(* Logix 5000 project; controller Machine_Smothies_V0 vendor 1 type 14 code 149 rev 36.11; software revision 36.00 *)

TASK MainTask (continuous, watchdog 500 ms) : MainProgram

MODULES
   Local : vendor 1 type 14 code 149 (Compact 0, rev 36.11)
      Discrete_IO : Embedded (Compact 1, rev 3.1, Output RPI 20 ms)
END_MODULES

VAR_GLOBAL   (* controller tags *)
   Acai : BOOL;
   Acai_Quant_1 : BOOL;
   Acai_Quant_2 : BOOL;
   Acai_Quant_3 : BOOL;
   Ajouter_Verre_Grand : BOOL;
   Ajouter_Verre_Moyen : BOOL;
   Ajouter_Verre_Petit : BOOL;
   Annuler_Base : BOOL;
   Annuler_Choix_Verre : BOOL;
   Annuler_Fruits : BOOL;
   Annuler_Lait : BOOL;
   Annuler_Sucrer : BOOL;
   Annuler_Tout : BOOL;
   Application_Lait : BOOL;
   Application_Sucre : BOOL;
   Avocat : BOOL;
   Avocat_Quant_1 : BOOL;
   Avocat_Quant_2 : BOOL;
   Avocat_Quant_3 : BOOL;
   Banane : BOOL;
   Banane_Quant_1 : BOOL;
   Banane_Quant_2 : BOOL;
   Banane_Quant_3 : BOOL;
   Bleuet : BOOL;
   Bleuet_Quant_1 : BOOL;
   Bleuet_Quant_2 : BOOL;
   Bleuet_Quant_3 : BOOL;
   Capteu_Sucrer : BOOL;
   Capteur_Base : BOOL;
   Capteur_Fruits : BOOL;
   Capteur_Grand : BOOL;
   Capteur_Lait : BOOL;
   Capteur_Moyen : BOOL;
   Capteur_Petit : BOOL;
   Capteur_Preparer : BOOL;
   Capteur_Pret : BOOL := 1;
   Choix_Verre_Grand : BOOL;
   Choix_Verre_Moyen : BOOL;
   Choix_Verre_Petit : BOOL;
   Descente_Bras_Mixeur : BOOL;
   Descente_Verre_Grand : BOOL;
   Descente_Verre_Moyen : BOOL;
   Descente_Verre_Petit : BOOL;
   Fraise : BOOL;
   Fraise_Quant_1 : BOOL;
   Fraise_Quant_2 : BOOL;
   Fraise_Quant_3 : BOOL;
   Framboise : BOOL;
   Framboise_Quant_1 : BOOL;
   Framboise_Quant_2 : BOOL;
   Framboise_Quant_3 : BOOL;
   Fruits_Champ : BOOL;
   Fruits_Champ_Quant_1 : BOOL;
   Fruits_Champ_Quant_2 : BOOL;
   Fruits_Champ_Quant_3 : BOOL;
   Fruits_Moine : BOOL;
   Fruits_Moine_Quant_1 : BOOL;
   Fruits_Moine_Quant_2 : BOOL;
   Fruits_Moine_Quant_3 : BOOL;
   Lait_Avoine : BOOL;
   Lait_Cajou : BOOL;
   Lait_Coco : BOOL;
   Lait_Soya : BOOL;
   Lait_Vache : BOOL;
   Lampe_Annuler_Base : BOOL;
   Lampe_Annuler_Choix_Verre : BOOL;
   Lampe_Annuler_Fruits : BOOL;
   Lampe_Annuler_Lait : BOOL;
   Lampe_Annuler_Sucrer : BOOL;
   Lampe_Annuler_Tout : BOOL;
   Lampe_Choix_Verre_Grand : BOOL;
   Lampe_Choix_Verre_Moyen : BOOL;
   Lampe_Choix_Verre_Petit : BOOL;
   Lampe_Lait_Avoine : BOOL;
   Lampe_Lait_Cajou : BOOL;
   Lampe_Lait_Coco : BOOL;
   Lampe_Lait_Soya : BOOL;
   Lampe_Lait_Vache : BOOL;
   Lampe_Non_Sucre : BOOL;
   Lampe_ON_OFF : BOOL;
   Lampe_Preparer : BOOL;
   Miel : BOOL;
   Miel_Quant_1 : BOOL;
   Miel_Quant_2 : BOOL;
   Miel_Quant_3 : BOOL;
   Mixer : BOOL;
   Non_Sucre : BOOL;
   ON_OFF : BOOL := 1;
   Peche : BOOL;
   Peche_Quant_1 : BOOL;
   Peche_Quant_2 : BOOL;
   Peche_Quant_3 : BOOL;
   Preparer : BOOL;
   Sucre : BOOL;
   Sucre_Quant_1 : BOOL;
   Sucre_Quant_2 : BOOL;
   Sucre_Quant_3 : BOOL;
   Tapis : BOOL;
   Tapis_ON_COND_INIT : BOOL;
   Xylitol : BOOL;
   Xylitol_Quant_1 : BOOL;
   Xylitol_Quant_2 : BOOL;
   Xylitol_Quant_3 : BOOL;
END_VAR

PROGRAM MainProgram   (* main routine MainRoutine *)
VAR
   BOR_01 : FBD_BOOLEAN_OR;
   BOR_02 : FBD_BOOLEAN_OR;
   OSRI_01 : FBD_ONESHOT := (InputBit := 1);
   RESD_01 : DOMINANT_RESET;
   TOFR_01 : FBD_TIMER := (PRE := 15000, ACC := 15000);
END_VAR

ROUTINE condition_initial   (* function block diagram *)
   SHEET 1
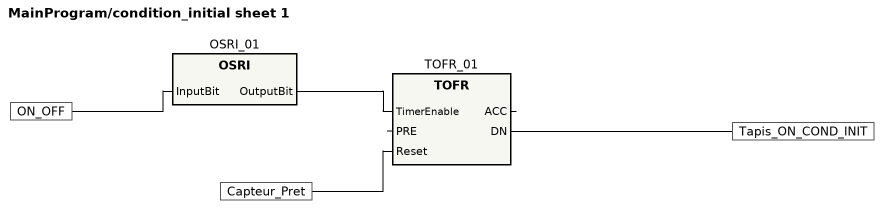
   OSRI_01 : OSRI(InputBit := ON_OFF);
   TOFR_01 : TOFR(TimerEnable := OSRI_01.OutputBit, Reset := Capteur_Pret);   // unwired pins: PRE ACC
   Tapis_ON_COND_INIT := TOFR_01.DN;
END_ROUTINE

ROUTINE MainRoutine   (* ladder *)
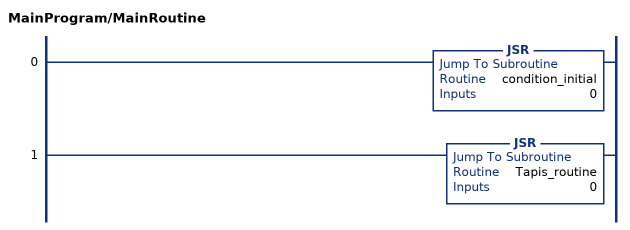
   0: JSR(condition_initial,0);
   1: JSR(Tapis_routine,0);
END_ROUTINE

ROUTINE Tapis_routine   (* function block diagram *)
   SHEET 1
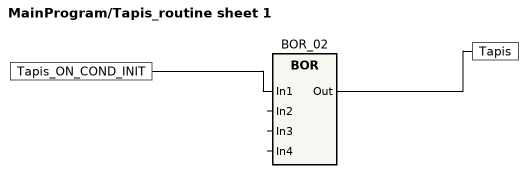
   BOR_02 : BOR(In1 := Tapis_ON_COND_INIT);   // unwired pins: In2 In3 In4
   Tapis := BOR_02.Out;
END_ROUTINE
END_PROGRAM
